TYPE T_CodeURL : STRING[20];
END_TYPE

(* stored: Version 1.1.0.1
   DUT T_CodeURL: Id {58fadf61-c751-407d-8f83-7ca26b4200c5} *)
